Yaskawa INFORM job: TEST_FIRST_LAYER_ARC.JBI

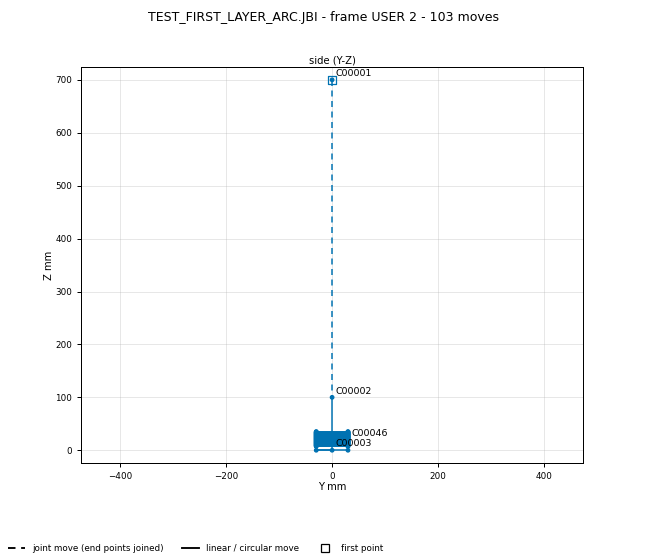
[picture p0: tool path of TEST_FIRST_LAYER_ARC.JBI in frame USER 2, 103 of 105 moves have a stored position in this frame; points joined in program order, loops and branches not executed]
/JOB
//NAME TEST_FIRST_LAYER_ARC
//POS
///NPOS 105,0,105,0,0,0
///USER 1
///TOOL 0
///POSTYPE USER
///RECTAN
///RCONF 1,0,0,0,0,0,0,0,0,0,0,0,0,0,0,0,0,0,0,0,0,0,0,0
C00000=1600.000,0.000,729.660,180.000,-50.000,0.000
///USER 2
///POSTYPE USER
///RECTAN
C00001=0.000,0.000,700.000,-180.000,-30.000,-45.000
C00002=0.000,0.000,100.000,-180.000,-0.000,-45.000
C00003=0.000,0.000,0.000,-180.000,0.000,-45.000
C00004=0.000,-30.000,0.000,-180.000,0.000,-45.000
C00005=0.000,30.000,0.000,-180.000,0.000,-45.000
C00006=0.000,30.000,7.380,-180.000,0.000,-45.000
C00007=0.000,-30.000,7.380,-180.000,0.000,-45.000
C00008=0.000,-30.000,7.960,-180.000,0.000,-45.000
C00009=0.000,30.000,7.960,-180.000,0.000,-45.000
C00010=0.000,30.000,8.540,-180.000,0.000,-45.000
C00011=0.000,-30.000,8.540,-180.000,0.000,-45.000
C00012=0.000,-30.000,9.120,-180.000,0.000,-45.000
C00013=0.000,30.000,9.120,-180.000,0.000,-45.000
C00014=0.000,30.000,9.700,-180.000,0.000,-45.000
C00015=0.000,-30.000,9.700,-180.000,0.000,-45.000
C00016=0.000,-30.000,10.280,-180.000,0.000,-45.000
C00017=0.000,30.000,10.280,-180.000,0.000,-45.000
C00018=0.000,30.000,10.860,-180.000,0.000,-45.000
C00019=0.000,-30.000,10.860,-180.000,0.000,-45.000
C00020=0.000,-30.000,11.440,-180.000,0.000,-45.000
C00021=0.000,30.000,11.440,-180.000,0.000,-45.000
C00022=0.000,30.000,12.020,-180.000,0.000,-45.000
C00023=0.000,-30.000,12.020,-180.000,0.000,-45.000
C00024=0.000,-30.000,12.600,-180.000,0.000,-45.000
C00025=0.000,30.000,12.600,-180.000,0.000,-45.000
C00026=0.000,30.000,13.180,-180.000,0.000,-45.000
C00027=0.000,-30.000,13.180,-180.000,0.000,-45.000
C00028=0.000,-30.000,13.760,-180.000,0.000,-45.000
C00029=0.000,30.000,13.760,-180.000,0.000,-45.000
C00030=0.000,30.000,14.340,-180.000,0.000,-45.000
C00031=0.000,-30.000,14.340,-180.000,0.000,-45.000
C00032=0.000,-30.000,14.920,-180.000,0.000,-45.000
C00033=0.000,30.000,14.920,-180.000,0.000,-45.000
C00034=0.000,30.000,15.500,-180.000,0.000,-45.000
C00035=0.000,-30.000,15.500,-180.000,0.000,-45.000
C00036=0.000,-30.000,16.080,-180.000,0.000,-45.000
C00037=0.000,30.000,16.080,-180.000,0.000,-45.000
C00038=0.000,30.000,16.660,-180.000,0.000,-45.000
C00039=0.000,-30.000,16.660,-180.000,0.000,-45.000
C00040=0.000,-30.000,17.240,-180.000,0.000,-45.000
C00041=0.000,30.000,17.240,-180.000,0.000,-45.000
C00042=0.000,30.000,17.820,-180.000,0.000,-45.000
C00043=0.000,-30.000,17.820,-180.000,0.000,-45.000
C00044=0.000,-30.000,18.400,-180.000,0.000,-45.000
C00045=0.000,30.000,18.400,-180.000,0.000,-45.000
C00046=0.000,30.000,18.980,-180.000,0.000,-45.000
C00047=0.000,-30.000,18.980,-180.000,0.000,-45.000
C00048=0.000,-30.000,19.560,-180.000,0.000,-45.000
C00049=0.000,30.000,19.560,-180.000,0.000,-45.000
C00050=0.000,30.000,20.140,-180.000,0.000,-45.000
C00051=0.000,-30.000,20.140,-180.000,0.000,-45.000
C00052=0.000,-30.000,20.720,-180.000,0.000,-45.000
C00053=0.000,30.000,20.720,-180.000,0.000,-45.000
C00054=0.000,30.000,21.300,-180.000,0.000,-45.000
C00055=0.000,-30.000,21.300,-180.000,0.000,-45.000
C00056=0.000,-30.000,21.880,-180.000,0.000,-45.000
C00057=0.000,30.000,21.880,-180.000,0.000,-45.000
C00058=0.000,30.000,22.460,-180.000,0.000,-45.000
C00059=0.000,-30.000,22.460,-180.000,0.000,-45.000
C00060=0.000,-30.000,23.040,-180.000,0.000,-45.000
C00061=0.000,30.000,23.040,-180.000,0.000,-45.000
C00062=0.000,30.000,23.620,-180.000,0.000,-45.000
C00063=0.000,-30.000,23.620,-180.000,0.000,-45.000
C00064=0.000,-30.000,24.200,-180.000,0.000,-45.000
C00065=0.000,30.000,24.200,-180.000,0.000,-45.000
C00066=0.000,30.000,24.780,-180.000,0.000,-45.000
C00067=0.000,-30.000,24.780,-180.000,0.000,-45.000
C00068=0.000,-30.000,25.360,-180.000,0.000,-45.000
C00069=0.000,30.000,25.360,-180.000,0.000,-45.000
C00070=0.000,30.000,25.940,-180.000,0.000,-45.000
C00071=0.000,-30.000,25.940,-180.000,0.000,-45.000
C00072=0.000,-30.000,26.520,-180.000,0.000,-45.000
C00073=0.000,30.000,26.520,-180.000,0.000,-45.000
C00074=0.000,30.000,27.100,-180.000,0.000,-45.000
C00075=0.000,-30.000,27.100,-180.000,0.000,-45.000
C00076=0.000,-30.000,27.680,-180.000,0.000,-45.000
C00077=0.000,30.000,27.680,-180.000,0.000,-45.000
C00078=0.000,30.000,28.260,-180.000,0.000,-45.000
C00079=0.000,-30.000,28.260,-180.000,0.000,-45.000
C00080=0.000,-30.000,28.840,-180.000,0.000,-45.000
C00081=0.000,30.000,28.840,-180.000,0.000,-45.000
C00082=0.000,30.000,29.420,-180.000,0.000,-45.000
C00083=0.000,-30.000,29.420,-180.000,0.000,-45.000
C00084=0.000,-30.000,30.000,-180.000,0.000,-45.000
C00085=0.000,30.000,30.000,-180.000,0.000,-45.000
C00086=0.000,30.000,30.580,-180.000,0.000,-45.000
C00087=0.000,-30.000,30.580,-180.000,0.000,-45.000
C00088=0.000,-30.000,31.160,-180.000,0.000,-45.000
C00089=0.000,30.000,31.160,-180.000,0.000,-45.000
C00090=0.000,30.000,31.740,-180.000,0.000,-45.000
C00091=0.000,-30.000,31.740,-180.000,0.000,-45.000
C00092=0.000,-30.000,32.320,-180.000,0.000,-45.000
C00093=0.000,30.000,32.320,-180.000,0.000,-45.000
C00094=0.000,30.000,32.900,-180.000,0.000,-45.000
C00095=0.000,-30.000,32.900,-180.000,0.000,-45.000
C00096=0.000,-30.000,33.480,-180.000,0.000,-45.000
C00097=0.000,30.000,33.480,-180.000,0.000,-45.000
C00098=0.000,30.000,34.060,-180.000,0.000,-45.000
C00099=0.000,-30.000,34.060,-180.000,0.000,-45.000
C00100=0.000,-30.000,34.640,-180.000,0.000,-45.000
C00101=0.000,30.000,34.640,-180.000,0.000,-45.000
C00102=0.000,30.000,35.220,-180.000,0.000,-45.000
C00103=0.000,-30.000,35.220,-180.000,0.000,-45.000
///USER 1
///POSTYPE USER
///RECTAN
C00104=1600.000,0.000,729.660,180.000,-50.000,0.000
///POSTYPE PULSE
///PULSE
EC00000=-29914,247808
EC00001=-29914,247808
EC00002=-29914,247808
EC00003=-29914,247808
EC00004=-29914,247808
EC00005=-29914,247808
EC00006=-29914,247808
EC00007=-29914,247808
EC00008=-29914,247808
EC00009=-29914,247808
EC00010=-29914,247808
EC00011=-29914,247808
EC00012=-29914,247808
EC00013=-29914,247808
EC00014=-29914,247808
EC00015=-29914,247808
EC00016=-29914,247808
EC00017=-29914,247808
EC00018=-29914,247808
EC00019=-29914,247808
EC00020=-29914,247808
EC00021=-29914,247808
EC00022=-29914,247808
EC00023=-29914,247808
EC00024=-29914,247808
EC00025=-29914,247808
EC00026=-29914,247808
EC00027=-29914,247808
EC00028=-29914,247808
EC00029=-29914,247808
EC00030=-29914,247808
EC00031=-29914,247808
EC00032=-29914,247808
EC00033=-29914,247808
EC00034=-29914,247808
EC00035=-29914,247808
EC00036=-29914,247808
EC00037=-29914,247808
EC00038=-29914,247808
EC00039=-29914,247808
EC00040=-29914,247808
EC00041=-29914,247808
EC00042=-29914,247808
EC00043=-29914,247808
EC00044=-29914,247808
EC00045=-29914,247808
EC00046=-29914,247808
EC00047=-29914,247808
EC00048=-29914,247808
EC00049=-29914,247808
EC00050=-29914,247808
EC00051=-29914,247808
EC00052=-29914,247808
EC00053=-29914,247808
EC00054=-29914,247808
EC00055=-29914,247808
EC00056=-29914,247808
EC00057=-29914,247808
EC00058=-29914,247808
EC00059=-29914,247808
EC00060=-29914,247808
EC00061=-29914,247808
EC00062=-29914,247808
EC00063=-29914,247808
EC00064=-29914,247808
EC00065=-29914,247808
EC00066=-29914,247808
EC00067=-29914,247808
EC00068=-29914,247808
EC00069=-29914,247808
EC00070=-29914,247808
EC00071=-29914,247808
EC00072=-29914,247808
EC00073=-29914,247808
EC00074=-29914,247808
EC00075=-29914,247808
EC00076=-29914,247808
EC00077=-29914,247808
EC00078=-29914,247808
EC00079=-29914,247808
EC00080=-29914,247808
EC00081=-29914,247808
EC00082=-29914,247808
EC00083=-29914,247808
EC00084=-29914,247808
EC00085=-29914,247808
EC00086=-29914,247808
EC00087=-29914,247808
EC00088=-29914,247808
EC00089=-29914,247808
EC00090=-29914,247808
EC00091=-29914,247808
EC00092=-29914,247808
EC00093=-29914,247808
EC00094=-29914,247808
EC00095=-29914,247808
EC00096=-29914,247808
EC00097=-29914,247808
EC00098=-29914,247808
EC00099=-29914,247808
EC00100=-29914,247808
EC00101=-29914,247808
EC00102=-29914,247808
EC00103=-29914,247808
EC00104=-29914,247808
//INST
///DATE 2022/12/08 12:43
///ATTR SC,RW,RJ
////FRAME USER 1
///GROUP1 RB1
///GROUP2 ST1
NOP
MOVJ C00000 VJ=25.00 PL=0 +MOVJ EC00000
MOVJ C00001 VJ=25.00 PL=0 +MOVJ EC00001
MOVJ C00002 VJ=25.00 PL=0 +MOVJ EC00002
SMOVL C00003 V=50.0 PL=0 +MOVJ EC00003
SMOVL C00004 V=50.0 PL=0 +MOVJ EC00004
ARCON ASF#(5)
SMOVL C00005 V=25.0 PL=0 +MOVJ EC00005
ARCOF AEF#(1)
CALL JOB:NOBUTTON10
SMOVL C00006 V=50.0 PL=0 +MOVJ EC00006
ARCON ASF#(5)
SMOVL C00007 V=25.0 PL=0 +MOVJ EC00007
ARCOF AEF#(1)
CALL JOB:NOBUTTON10
SMOVL C00008 V=50.0 PL=0 +MOVJ EC00008
ARCON ASF#(5)
SMOVL C00009 V=25.0 PL=0 +MOVJ EC00009
ARCOF AEF#(1)
CALL JOB:NOBUTTON10
SMOVL C00010 V=50.0 PL=0 +MOVJ EC00010
ARCON ASF#(5)
SMOVL C00011 V=25.0 PL=0 +MOVJ EC00011
ARCOF AEF#(1)
CALL JOB:NOBUTTON10
SMOVL C00012 V=50.0 PL=0 +MOVJ EC00012
ARCON ASF#(5)
SMOVL C00013 V=25.0 PL=0 +MOVJ EC00013
ARCOF AEF#(1)
CALL JOB:NOBUTTON10
SMOVL C00014 V=50.0 PL=0 +MOVJ EC00014
ARCON ASF#(5)
SMOVL C00015 V=25.0 PL=0 +MOVJ EC00015
ARCOF AEF#(1)
CALL JOB:NOBUTTON10
SMOVL C00016 V=50.0 PL=0 +MOVJ EC00016
ARCON ASF#(5)
SMOVL C00017 V=25.0 PL=0 +MOVJ EC00017
ARCOF AEF#(1)
CALL JOB:NOBUTTON10
SMOVL C00018 V=50.0 PL=0 +MOVJ EC00018
ARCON ASF#(5)
SMOVL C00019 V=25.0 PL=0 +MOVJ EC00019
ARCOF AEF#(1)
CALL JOB:NOBUTTON10
SMOVL C00020 V=50.0 PL=0 +MOVJ EC00020
ARCON ASF#(5)
SMOVL C00021 V=25.0 PL=0 +MOVJ EC00021
ARCOF AEF#(1)
CALL JOB:NOBUTTON10
SMOVL C00022 V=50.0 PL=0 +MOVJ EC00022
ARCON ASF#(5)
SMOVL C00023 V=25.0 PL=0 +MOVJ EC00023
ARCOF AEF#(1)
CALL JOB:NOBUTTON10
SMOVL C00024 V=50.0 PL=0 +MOVJ EC00024
ARCON ASF#(5)
SMOVL C00025 V=25.0 PL=0 +MOVJ EC00025
ARCOF AEF#(1)
CALL JOB:NOBUTTON10
SMOVL C00026 V=50.0 PL=0 +MOVJ EC00026
ARCON ASF#(5)
SMOVL C00027 V=25.0 PL=0 +MOVJ EC00027
ARCOF AEF#(1)
CALL JOB:NOBUTTON10
SMOVL C00028 V=50.0 PL=0 +MOVJ EC00028
ARCON ASF#(5)
SMOVL C00029 V=25.0 PL=0 +MOVJ EC00029
ARCOF AEF#(1)
CALL JOB:NOBUTTON10
SMOVL C00030 V=50.0 PL=0 +MOVJ EC00030
ARCON ASF#(5)
SMOVL C00031 V=25.0 PL=0 +MOVJ EC00031
ARCOF AEF#(1)
CALL JOB:NOBUTTON10
SMOVL C00032 V=50.0 PL=0 +MOVJ EC00032
ARCON ASF#(5)
SMOVL C00033 V=25.0 PL=0 +MOVJ EC00033
ARCOF AEF#(1)
CALL JOB:NOBUTTON10
SMOVL C00034 V=50.0 PL=0 +MOVJ EC00034
ARCON ASF#(5)
SMOVL C00035 V=25.0 PL=0 +MOVJ EC00035
ARCOF AEF#(1)
CALL JOB:NOBUTTON10
SMOVL C00036 V=50.0 PL=0 +MOVJ EC00036
ARCON ASF#(5)
SMOVL C00037 V=25.0 PL=0 +MOVJ EC00037
ARCOF AEF#(1)
CALL JOB:NOBUTTON10
SMOVL C00038 V=50.0 PL=0 +MOVJ EC00038
ARCON ASF#(5)
SMOVL C00039 V=25.0 PL=0 +MOVJ EC00039
ARCOF AEF#(1)
CALL JOB:NOBUTTON10
SMOVL C00040 V=50.0 PL=0 +MOVJ EC00040
ARCON ASF#(5)
SMOVL C00041 V=25.0 PL=0 +MOVJ EC00041
ARCOF AEF#(1)
CALL JOB:NOBUTTON10
SMOVL C00042 V=50.0 PL=0 +MOVJ EC00042
ARCON ASF#(5)
SMOVL C00043 V=25.0 PL=0 +MOVJ EC00043
ARCOF AEF#(1)
CALL JOB:NOBUTTON10
SMOVL C00044 V=50.0 PL=0 +MOVJ EC00044
ARCON ASF#(5)
SMOVL C00045 V=25.0 PL=0 +MOVJ EC00045
ARCOF AEF#(1)
CALL JOB:NOBUTTON10
SMOVL C00046 V=50.0 PL=0 +MOVJ EC00046
ARCON ASF#(5)
SMOVL C00047 V=25.0 PL=0 +MOVJ EC00047
ARCOF AEF#(1)
CALL JOB:NOBUTTON10
SMOVL C00048 V=50.0 PL=0 +MOVJ EC00048
ARCON ASF#(5)
SMOVL C00049 V=25.0 PL=0 +MOVJ EC00049
ARCOF AEF#(1)
CALL JOB:NOBUTTON10
SMOVL C00050 V=50.0 PL=0 +MOVJ EC00050
ARCON ASF#(5)
SMOVL C00051 V=25.0 PL=0 +MOVJ EC00051
ARCOF AEF#(1)
CALL JOB:NOBUTTON10
SMOVL C00052 V=50.0 PL=0 +MOVJ EC00052
ARCON ASF#(5)
SMOVL C00053 V=25.0 PL=0 +MOVJ EC00053
ARCOF AEF#(1)
CALL JOB:NOBUTTON10
SMOVL C00054 V=50.0 PL=0 +MOVJ EC00054
ARCON ASF#(5)
SMOVL C00055 V=25.0 PL=0 +MOVJ EC00055
ARCOF AEF#(1)
CALL JOB:NOBUTTON10
SMOVL C00056 V=50.0 PL=0 +MOVJ EC00056
ARCON ASF#(5)
SMOVL C00057 V=25.0 PL=0 +MOVJ EC00057
ARCOF AEF#(1)
CALL JOB:NOBUTTON10
SMOVL C00058 V=50.0 PL=0 +MOVJ EC00058
ARCON ASF#(5)
SMOVL C00059 V=25.0 PL=0 +MOVJ EC00059
ARCOF AEF#(1)
CALL JOB:NOBUTTON10
SMOVL C00060 V=50.0 PL=0 +MOVJ EC00060
ARCON ASF#(5)
SMOVL C00061 V=25.0 PL=0 +MOVJ EC00061
ARCOF AEF#(1)
CALL JOB:NOBUTTON10
SMOVL C00062 V=50.0 PL=0 +MOVJ EC00062
ARCON ASF#(5)
SMOVL C00063 V=25.0 PL=0 +MOVJ EC00063
ARCOF AEF#(1)
CALL JOB:NOBUTTON10
SMOVL C00064 V=50.0 PL=0 +MOVJ EC00064
ARCON ASF#(5)
SMOVL C00065 V=25.0 PL=0 +MOVJ EC00065
ARCOF AEF#(1)
CALL JOB:NOBUTTON10
SMOVL C00066 V=50.0 PL=0 +MOVJ EC00066
ARCON ASF#(5)
SMOVL C00067 V=25.0 PL=0 +MOVJ EC00067
ARCOF AEF#(1)
CALL JOB:NOBUTTON10
SMOVL C00068 V=50.0 PL=0 +MOVJ EC00068
ARCON ASF#(5)
SMOVL C00069 V=25.0 PL=0 +MOVJ EC00069
ARCOF AEF#(1)
CALL JOB:NOBUTTON10
SMOVL C00070 V=50.0 PL=0 +MOVJ EC00070
ARCON ASF#(5)
SMOVL C00071 V=25.0 PL=0 +MOVJ EC00071
ARCOF AEF#(1)
CALL JOB:NOBUTTON10
SMOVL C00072 V=50.0 PL=0 +MOVJ EC00072
ARCON ASF#(5)
SMOVL C00073 V=25.0 PL=0 +MOVJ EC00073
ARCOF AEF#(1)
CALL JOB:NOBUTTON10
SMOVL C00074 V=50.0 PL=0 +MOVJ EC00074
ARCON ASF#(5)
SMOVL C00075 V=25.0 PL=0 +MOVJ EC00075
ARCOF AEF#(1)
CALL JOB:NOBUTTON10
SMOVL C00076 V=50.0 PL=0 +MOVJ EC00076
ARCON ASF#(5)
SMOVL C00077 V=25.0 PL=0 +MOVJ EC00077
ARCOF AEF#(1)
CALL JOB:NOBUTTON10
SMOVL C00078 V=50.0 PL=0 +MOVJ EC00078
ARCON ASF#(5)
SMOVL C00079 V=25.0 PL=0 +MOVJ EC00079
ARCOF AEF#(1)
CALL JOB:NOBUTTON10
SMOVL C00080 V=50.0 PL=0 +MOVJ EC00080
ARCON ASF#(5)
SMOVL C00081 V=25.0 PL=0 +MOVJ EC00081
ARCOF AEF#(1)
CALL JOB:NOBUTTON10
SMOVL C00082 V=50.0 PL=0 +MOVJ EC00082
ARCON ASF#(5)
SMOVL C00083 V=25.0 PL=0 +MOVJ EC00083
ARCOF AEF#(1)
CALL JOB:NOBUTTON10
SMOVL C00084 V=50.0 PL=0 +MOVJ EC00084
ARCON ASF#(5)
SMOVL C00085 V=25.0 PL=0 +MOVJ EC00085
ARCOF AEF#(1)
CALL JOB:NOBUTTON10
SMOVL C00086 V=50.0 PL=0 +MOVJ EC00086
ARCON ASF#(5)
SMOVL C00087 V=25.0 PL=0 +MOVJ EC00087
ARCOF AEF#(1)
CALL JOB:NOBUTTON10
SMOVL C00088 V=50.0 PL=0 +MOVJ EC00088
ARCON ASF#(5)
SMOVL C00089 V=25.0 PL=0 +MOVJ EC00089
ARCOF AEF#(1)
CALL JOB:NOBUTTON10
SMOVL C00090 V=50.0 PL=0 +MOVJ EC00090
ARCON ASF#(5)
SMOVL C00091 V=25.0 PL=0 +MOVJ EC00091
ARCOF AEF#(1)
CALL JOB:NOBUTTON10
SMOVL C00092 V=50.0 PL=0 +MOVJ EC00092
ARCON ASF#(5)
SMOVL C00093 V=25.0 PL=0 +MOVJ EC00093
ARCOF AEF#(1)
CALL JOB:NOBUTTON10
SMOVL C00094 V=50.0 PL=0 +MOVJ EC00094
ARCON ASF#(5)
SMOVL C00095 V=25.0 PL=0 +MOVJ EC00095
ARCOF AEF#(1)
CALL JOB:NOBUTTON10
SMOVL C00096 V=50.0 PL=0 +MOVJ EC00096
ARCON ASF#(5)
SMOVL C00097 V=25.0 PL=0 +MOVJ EC00097
ARCOF AEF#(1)
CALL JOB:NOBUTTON10
SMOVL C00098 V=50.0 PL=0 +MOVJ EC00098
ARCON ASF#(5)
SMOVL C00099 V=25.0 PL=0 +MOVJ EC00099
ARCOF AEF#(1)
CALL JOB:NOBUTTON10
SMOVL C00100 V=50.0 PL=0 +MOVJ EC00100
ARCON ASF#(5)
SMOVL C00101 V=25.0 PL=0 +MOVJ EC00101
ARCOF AEF#(1)
CALL JOB:NOBUTTON10
SMOVL C00102 V=50.0 PL=0 +MOVJ EC00102
ARCON ASF#(5)
SMOVL C00103 V=25.0 PL=0 +MOVJ EC00103
ARCOF AEF#(1)
CALL JOB:NOBUTTON10
MOVJ C00104 VJ=25.00 PL=0 +MOVJ EC00104
END
